SUBAPPLICATION AX_2_2 (* AX_OR and AX_SPLIT for a 2-to-2 Connection *)
  (* Standard: 61499-2 *)
  (* Version 1.0, 2026-05-29, franz, Meisterschulen am Ostbahnhof *)
  (* Documentation:
  2 AX-Quellen ODER-verknüpft auf 2 AX-Ziele verteilt
   Kombiniert AX_OR_2 und AX_SPLIT_2 zu einem fertigen Baustein: nimmt IN1/IN2 entgegen, verknüpft beide per ODER zu einem gemeinsamen Signal und verteilt dieses anschließend auf OUT1/OUT2.
   Typischer Einsatz: mehrere Bedienelemente (z.B. SoftKey und Aux-Taster) sollen gemeinsam mehrere Ziele ansteuern (z.B. einen Ausgang UND eine Hintergrundfarbe-SubApp), ohne AX_OR_2 und AX_SPLIT_2 jedes Mal einzeln zu verdrahten.
   Für andere Quellen-/Ziel-Anzahlen: AX_3_3 (3→3), AX_2_3 (2→3), AX_3_2 (3→2).
  *)
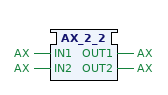
  SOCKETS
    IN1 : adapter::types::unidirectional::AX;
    IN2 : adapter::types::unidirectional::AX;
  END_SOCKETS
  PLUGS
    OUT1 : adapter::types::unidirectional::AX;
    OUT2 : adapter::types::unidirectional::AX;
  END_PLUGS
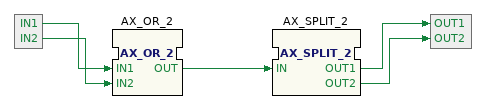
  FBS
    AX_SPLIT_2 : adapter::events::unidirectional::AX_SPLIT_2;
    AX_OR_2 : adapter::booleanOperators::AX_OR_2;
  END_FBS
  ADAPTER_CONNECTIONS
    AX_OR_2.OUT TO AX_SPLIT_2.IN;
    AX_SPLIT_2.OUT1 TO OUT1;
    AX_SPLIT_2.OUT2 TO OUT2;
    IN1 TO AX_OR_2.IN1;
    IN2 TO AX_OR_2.IN2;
  END_CONNECTIONS
END_SUBAPPLICATION
